{attribute 'TcGenerated'}
{attribute 'no-analysis'}
{attribute 'linkalways'}
// This function has been automatically generated from the project information.
VAR_GLOBAL CONSTANT
	{attribute 'const_non_replaced'}
	stLibVersion_snappy : ST_LibVersion := (iMajor := 0, iMinor := 3, iBuild := 1, iRevision := 0, nFlags := 0, sVersion := '0.3.3.0');
END_VAR

(* stored: Version 1.1.0.1, ProductVersion 3.1.4024.13
   GVL Global_Version: Id {e8c1b537-7c98-47f8-8420-3bfa56237b19} *)
